VAR_GLOBAL
	DefaultLogger : T_Logger;
END_VAR

(* stored: Version 1.1.0.1, ProductVersion 3.1.4024.15
   GVL Globals: Id {3c6e8760-3da3-4725-ba68-f667404cea96} *)
